FUNCTION F_SendUDPMessage : HRESULT
VAR_INPUT
    psMessage			:	POINTER TO STRING;
    fbSocket			:	REFERENCE TO FB_ConnectionlessSocket;
    sHost				:	STRING;
    nPort				:	UINT;
END_VAR

VAR
    fbSend				:	FB_SocketUdpSendTo;
END_VAR

IF psMessage <> 0 AND __ISVALIDREF(fbSocket) THEN
    fbSend.hSocket		:= fbSocket.hSocket;
    fbSend.sRemoteHost	:= sHost;
    fbSend.nRemotePort	:= nPort;
    fbSend.pSrc 		:= psMessage;
    fbSend.cbLen		:= LEN2(psMessage);
    fbSend.bExecute	 	:= TRUE;
    fbSend();

    fbSend.bExecute 	R= fbSend.bBusy;
END_IF

END_FUNCTION

(* stored: Version 1.1.0.1
   POU F_SendUDPMessage: Id {6df3303a-af20-4404-b690-e252d379813c}, SpecialFunc None *)
